FUNCTION_BLOCK B_1Event_5States_Unreachable (* Basic FB with empty ECC *)
  (* Standard: 61499-2 *)
  (* Version 1.0, 2023-09-22, AK124910 *)
  PACKAGE servSeq;
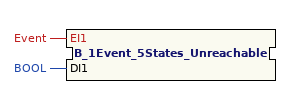
  EVENT_INPUT
    EI1;
  END_EVENT
  VAR_INPUT
    DI1 : BOOL;
  END_VAR
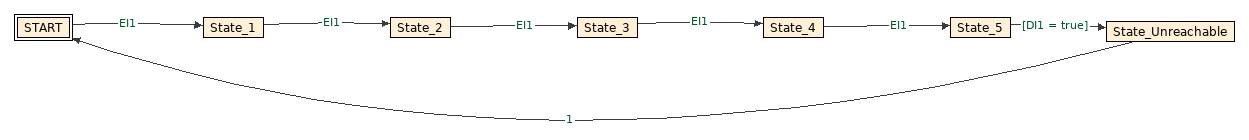
  EC_STATES
    START; (* Initial State *)
    State_1;
    State_2;
    State_3;
    State_4;
    State_5;
    State_Unreachable;
  END_STATES
  EC_TRANSITIONS
    START TO State_1 := EI1;
    State_1 TO State_2 := EI1;
    State_2 TO State_3 := EI1;
    State_3 TO State_4 := EI1;
    State_4 TO State_5 := EI1;
    State_5 TO State_Unreachable := [DI1 = true];
    State_Unreachable TO START := 1;
  END_TRANSITIONS
  SERVICE external/internal_interface (* Basic FB with empty ECC *)
    SEQUENCE ServiceSequence (* Coverage: 0.14285715 *) {SET_ATTRIBUTE(StartState, START)}
      external.EI1();
    END_SEQUENCE
    SEQUENCE ServiceSequence_1 (* Coverage: 0.14285715 *) {SET_ATTRIBUTE(StartState, State_1)}
      external.EI1();
    END_SEQUENCE
    SEQUENCE ServiceSequence_2 (* Coverage: 0.14285715 *) {SET_ATTRIBUTE(StartState, State_2)}
      external.EI1();
    END_SEQUENCE
    SEQUENCE ServiceSequence_3 (* Coverage: 0.14285715 *) {SET_ATTRIBUTE(StartState, State_3)}
      external.EI1();
    END_SEQUENCE
    SEQUENCE ServiceSequence_4 (* Coverage: 0.14285715 *) {SET_ATTRIBUTE(StartState, State_4)}
      external.EI1();
    END_SEQUENCE
    SEQUENCE ServiceSequence_5 (* Coverage: 0.14285715 *) {SET_ATTRIBUTE(StartState, State_Unreachable)}
      external.EI1();
    END_SEQUENCE
  END_SERVICE
END_FUNCTION_BLOCK
